(* CoDeSys 2.3 export: SIMULATION.EXP *)

(* POU LAB/gateManage, CFC *)
PROGRAM gateManage
VAR
	gate18 : fbGateManage;
	gate4: fbGateManage;
	gate11: fbGateManage;
	gate17: fbGateManage;
	gate14: fbGateManage;
	gate5: fbGateManage;
	gate8: fbGateManage;
	gate7: fbGateManage;
	gate9: fbGateManage;
	gate10: fbGateManage;
	gate6: fbGateManage;
	wtrPump: fbPumpManage;
	olPump: fbPumpManage;
END_VAR
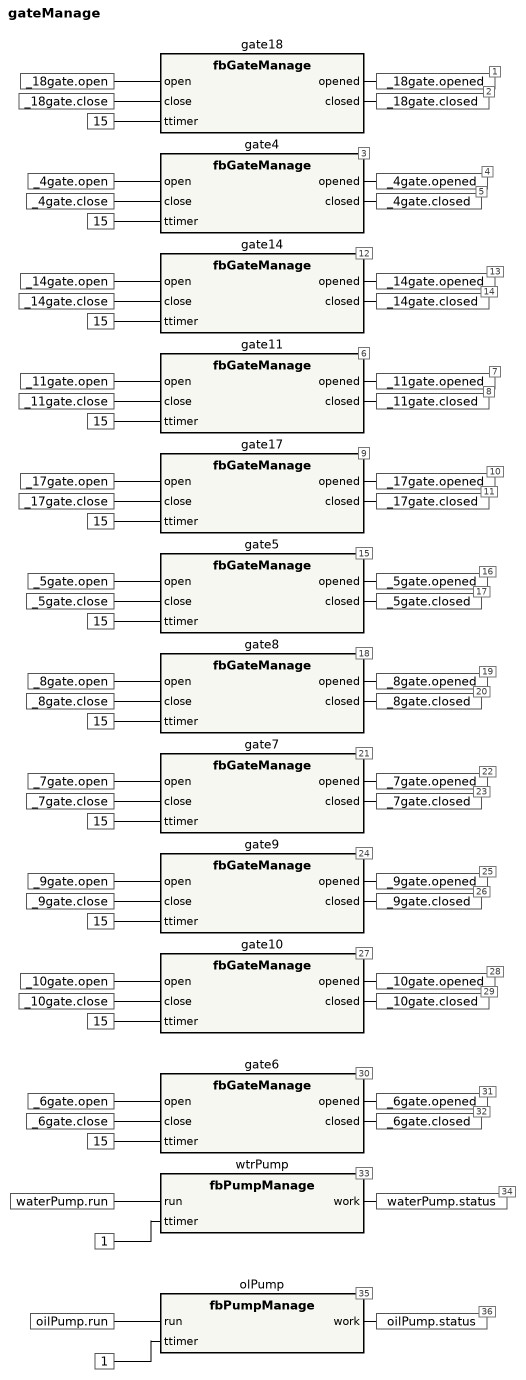
_CFC_ (* Continuous Function Chart, elements in execution order *)
#0 gate18:fbGateManage(open: _18gate.open, close: _18gate.close, ttimer: 15)
#1 _18gate.opened <= #0.opened
#2 _18gate.closed <= #0.closed
#3 gate4:fbGateManage(open: _4gate.open, close: _4gate.close, ttimer: 15)
#4 _4gate.opened <= #3.opened
#5 _4gate.closed <= #3.closed
#6 gate11:fbGateManage(open: _11gate.open, close: _11gate.close, ttimer: 15)
#7 _11gate.opened <= #6.opened
#8 _11gate.closed <= #6.closed
#9 gate17:fbGateManage(open: _17gate.open, close: _17gate.close, ttimer: 15)
#10 _17gate.opened <= #9.opened
#11 _17gate.closed <= #9.closed
#12 gate14:fbGateManage(open: _14gate.open, close: _14gate.close, ttimer: 15)
#13 _14gate.opened <= #12.opened
#14 _14gate.closed <= #12.closed
#15 gate5:fbGateManage(open: _5gate.open, close: _5gate.close, ttimer: 15)
#16 _5gate.opened <= #15.opened
#17 _5gate.closed <= #15.closed
#18 gate8:fbGateManage(open: _8gate.open, close: _8gate.close, ttimer: 15)
#19 _8gate.opened <= #18.opened
#20 _8gate.closed <= #18.closed
#21 gate7:fbGateManage(open: _7gate.open, close: _7gate.close, ttimer: 15)
#22 _7gate.opened <= #21.opened
#23 _7gate.closed <= #21.closed
#24 gate9:fbGateManage(open: _9gate.open, close: _9gate.close, ttimer: 15)
#25 _9gate.opened <= #24.opened
#26 _9gate.closed <= #24.closed
#27 gate10:fbGateManage(open: _10gate.open, close: _10gate.close, ttimer: 15)
#28 _10gate.opened <= #27.opened
#29 _10gate.closed <= #27.closed
#30 gate6:fbGateManage(open: _6gate.open, close: _6gate.close, ttimer: 15)
#31 _6gate.opened <= #30.opened
#32 _6gate.closed <= #30.closed
#33 wtrPump:fbPumpManage(run: waterPump.run, ttimer: 1)
#34 waterPump.status <= #33.work
#35 olPump:fbPumpManage(run: oilPump.run, ttimer: 1)
#36 oilPump.status <= #35.work
_END_CFC_
(* the same logic as Structured Text *)
gate18(open := _18gate.open, close := _18gate.close, ttimer := 15);
_18gate.opened := gate18.opened;
_18gate.closed := gate18.closed;
gate4(open := _4gate.open, close := _4gate.close, ttimer := 15);
_4gate.opened := gate4.opened;
_4gate.closed := gate4.closed;
gate11(open := _11gate.open, close := _11gate.close, ttimer := 15);
_11gate.opened := gate11.opened;
_11gate.closed := gate11.closed;
gate17(open := _17gate.open, close := _17gate.close, ttimer := 15);
_17gate.opened := gate17.opened;
_17gate.closed := gate17.closed;
gate14(open := _14gate.open, close := _14gate.close, ttimer := 15);
_14gate.opened := gate14.opened;
_14gate.closed := gate14.closed;
gate5(open := _5gate.open, close := _5gate.close, ttimer := 15);
_5gate.opened := gate5.opened;
_5gate.closed := gate5.closed;
gate8(open := _8gate.open, close := _8gate.close, ttimer := 15);
_8gate.opened := gate8.opened;
_8gate.closed := gate8.closed;
gate7(open := _7gate.open, close := _7gate.close, ttimer := 15);
_7gate.opened := gate7.opened;
_7gate.closed := gate7.closed;
gate9(open := _9gate.open, close := _9gate.close, ttimer := 15);
_9gate.opened := gate9.opened;
_9gate.closed := gate9.closed;
gate10(open := _10gate.open, close := _10gate.close, ttimer := 15);
_10gate.opened := gate10.opened;
_10gate.closed := gate10.closed;
gate6(open := _6gate.open, close := _6gate.close, ttimer := 15);
_6gate.opened := gate6.opened;
_6gate.closed := gate6.closed;
wtrPump(run := waterPump.run, ttimer := 1);
waterPump.status := wtrPump.work;
olPump(run := oilPump.run, ttimer := 1);
oilPump.status := olPump.work;
END_PROGRAM

(* POU LAB/fbGateManage, CFC *)
FUNCTION_BLOCK fbGateManage
VAR_INPUT
	open : BOOL;
	close : BOOL;
	ttimer : WORD;
END_VAR
VAR_OUTPUT
	opened : BOOL;
	closed : BOOL;
END_VAR
VAR
	t :TIME := T#20s;
	tOpen: TON;
	tClose: TON;
	OpenTON : TON;
END_VAR
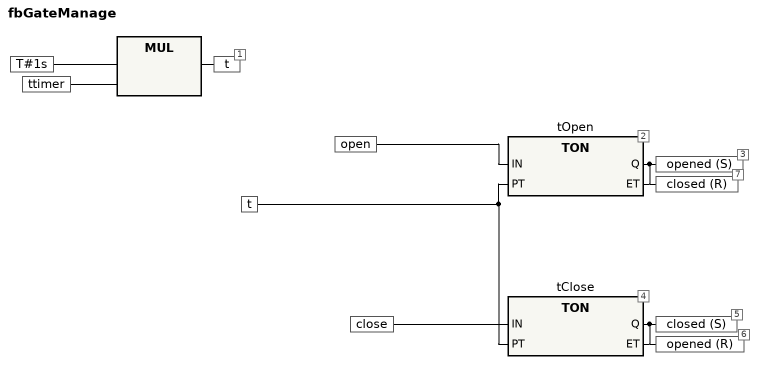
_CFC_ (* Continuous Function Chart, elements in execution order *)
#0 MUL(T#1s, ttimer)
#1 t <= #0
#2 tOpen:TON(IN: open, PT: t)
#3 S opened <= #2.Q
#4 tClose:TON(IN: close, PT: t)
#5 S closed <= #4.Q
#6 R opened <= #4.Q
#7 R closed <= #2.Q
_END_CFC_
(* the same logic as Structured Text *)
t := T#1s * ttimer;
tOpen(IN := open, PT := t);
IF tOpen.Q THEN opened := TRUE; END_IF;
tClose(IN := close, PT := t);
IF tClose.Q THEN closed := TRUE; END_IF;
IF tClose.Q THEN opened := FALSE; END_IF;
IF tOpen.Q THEN closed := FALSE; END_IF;
END_FUNCTION_BLOCK

(* POU LAB/fbPumpManage, CFC *)
FUNCTION_BLOCK fbPumpManage
VAR_INPUT
	run : BOOL;
	ttimer : WORD := 1;
END_VAR
VAR_OUTPUT
	work : BOOL;
END_VAR
VAR
	tOpen: TON;
	tClose: TON;
	trig: F_TRIG;
END_VAR
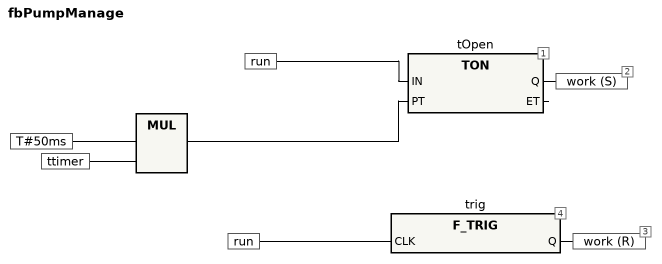
_CFC_ (* Continuous Function Chart, elements in execution order *)
#0 MUL(T#50ms, ttimer)
#1 tOpen:TON(IN: run, PT: #0)
#2 S work <= #1.Q
#3 R work <= #4.Q
#4 trig:F_TRIG(CLK: run)
_END_CFC_
(* the same logic as Structured Text *)
tOpen(IN := run, PT := T#50ms * ttimer);
IF tOpen.Q THEN work := TRUE; END_IF;
IF trig.Q THEN work := FALSE; END_IF;
trig(CLK := run);
END_FUNCTION_BLOCK
